TEXTLIST AxesPointingModelSetupPartsTextList
  0 = 'Part 1'
  1 = 'Part 2'
   = ''
END_TEXTLIST

(* stored: Version 1.1.0.1, ProductVersion 3.1.4018.5
   TextList AxesPointingModelSetupPartsTextList: Id {1a498288-bf27-46cb-bdcd-a65b4087d4da} *)
